FUNCTION_BLOCK ASSEMBLE_AW_FROM_AX (* this Function combines the 16 AX (BOOL) adapters to a AW (WORD) *)
  (* Standard: 61499-2; Description: Copyright (c) 2026 Meisterschulen am Ostbahnhof SPDX-License-Identifier: EPL-2.0 *)
  (* Version 1.0, 2026-05-16, Franz Höpfinger, Meisterschulen am Ostbahnhof, initial API and implementation and/or initial documentation *)
  PACKAGE adapter::assembling;
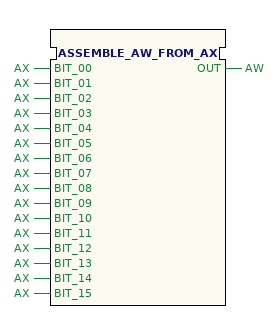
  SOCKETS
    BIT_00 : adapter::types::unidirectional::AX; (* Bool Bit 0 *)
    BIT_01 : adapter::types::unidirectional::AX; (* Bool Bit 1 *)
    BIT_02 : adapter::types::unidirectional::AX; (* Bool Bit 2 *)
    BIT_03 : adapter::types::unidirectional::AX; (* Bool Bit 3 *)
    BIT_04 : adapter::types::unidirectional::AX; (* Bool Bit 4 *)
    BIT_05 : adapter::types::unidirectional::AX; (* Bool Bit 5 *)
    BIT_06 : adapter::types::unidirectional::AX; (* Bool Bit 6 *)
    BIT_07 : adapter::types::unidirectional::AX; (* Bool Bit 7 *)
    BIT_08 : adapter::types::unidirectional::AX; (* Bool Bit 8 *)
    BIT_09 : adapter::types::unidirectional::AX; (* Bool Bit 9 *)
    BIT_10 : adapter::types::unidirectional::AX; (* Bool Bit 10 *)
    BIT_11 : adapter::types::unidirectional::AX; (* Bool Bit 11 *)
    BIT_12 : adapter::types::unidirectional::AX; (* Bool Bit 12 *)
    BIT_13 : adapter::types::unidirectional::AX; (* Bool Bit 13 *)
    BIT_14 : adapter::types::unidirectional::AX; (* Bool Bit 14 *)
    BIT_15 : adapter::types::unidirectional::AX; (* Bool Bit 15 *)
  END_SOCKETS
  PLUGS
    OUT : adapter::types::unidirectional::AW; (* WORD Output *)
  END_PLUGS
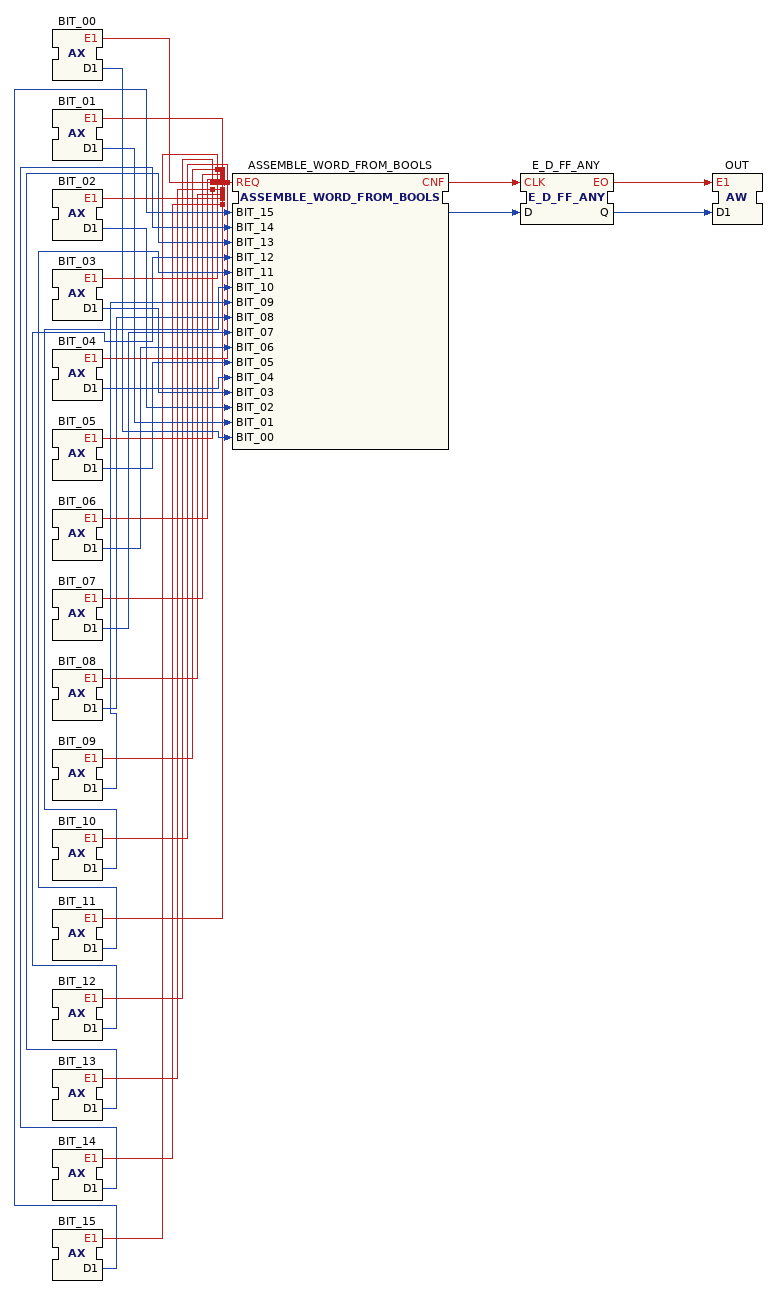
  FBS
    ASSEMBLE_WORD_FROM_BOOLS : eclipse4diac::utils::assembling::ASSEMBLE_WORD_FROM_BOOLS;
    E_D_FF_ANY : iec61499::events::E_D_FF_ANY;
  END_FBS
  EVENT_CONNECTIONS
    BIT_00.E1 TO ASSEMBLE_WORD_FROM_BOOLS.REQ;
    BIT_01.E1 TO ASSEMBLE_WORD_FROM_BOOLS.REQ;
    BIT_02.E1 TO ASSEMBLE_WORD_FROM_BOOLS.REQ;
    BIT_03.E1 TO ASSEMBLE_WORD_FROM_BOOLS.REQ;
    BIT_04.E1 TO ASSEMBLE_WORD_FROM_BOOLS.REQ;
    BIT_05.E1 TO ASSEMBLE_WORD_FROM_BOOLS.REQ;
    BIT_06.E1 TO ASSEMBLE_WORD_FROM_BOOLS.REQ;
    BIT_07.E1 TO ASSEMBLE_WORD_FROM_BOOLS.REQ;
    BIT_08.E1 TO ASSEMBLE_WORD_FROM_BOOLS.REQ;
    BIT_09.E1 TO ASSEMBLE_WORD_FROM_BOOLS.REQ;
    BIT_10.E1 TO ASSEMBLE_WORD_FROM_BOOLS.REQ;
    BIT_11.E1 TO ASSEMBLE_WORD_FROM_BOOLS.REQ;
    BIT_12.E1 TO ASSEMBLE_WORD_FROM_BOOLS.REQ;
    BIT_13.E1 TO ASSEMBLE_WORD_FROM_BOOLS.REQ;
    BIT_14.E1 TO ASSEMBLE_WORD_FROM_BOOLS.REQ;
    BIT_15.E1 TO ASSEMBLE_WORD_FROM_BOOLS.REQ;
    ASSEMBLE_WORD_FROM_BOOLS.CNF TO E_D_FF_ANY.CLK;
    E_D_FF_ANY.EO TO OUT.E1;
  END_CONNECTIONS
  DATA_CONNECTIONS
    ASSEMBLE_WORD_FROM_BOOLS. TO E_D_FF_ANY.D;
    E_D_FF_ANY.Q TO OUT.D1;
    BIT_15.D1 TO ASSEMBLE_WORD_FROM_BOOLS.BIT_15;
    BIT_14.D1 TO ASSEMBLE_WORD_FROM_BOOLS.BIT_14;
    BIT_13.D1 TO ASSEMBLE_WORD_FROM_BOOLS.BIT_13;
    BIT_12.D1 TO ASSEMBLE_WORD_FROM_BOOLS.BIT_12;
    BIT_11.D1 TO ASSEMBLE_WORD_FROM_BOOLS.BIT_11;
    BIT_10.D1 TO ASSEMBLE_WORD_FROM_BOOLS.BIT_10;
    BIT_09.D1 TO ASSEMBLE_WORD_FROM_BOOLS.BIT_09;
    BIT_08.D1 TO ASSEMBLE_WORD_FROM_BOOLS.BIT_08;
    BIT_07.D1 TO ASSEMBLE_WORD_FROM_BOOLS.BIT_07;
    BIT_06.D1 TO ASSEMBLE_WORD_FROM_BOOLS.BIT_06;
    BIT_05.D1 TO ASSEMBLE_WORD_FROM_BOOLS.BIT_05;
    BIT_04.D1 TO ASSEMBLE_WORD_FROM_BOOLS.BIT_04;
    BIT_03.D1 TO ASSEMBLE_WORD_FROM_BOOLS.BIT_03;
    BIT_02.D1 TO ASSEMBLE_WORD_FROM_BOOLS.BIT_02;
    BIT_01.D1 TO ASSEMBLE_WORD_FROM_BOOLS.BIT_01;
    BIT_00.D1 TO ASSEMBLE_WORD_FROM_BOOLS.BIT_00;
  END_CONNECTIONS
END_FUNCTION_BLOCK
